KUKA KRL data list: pick_from_playingfield.dat

&ACCESS RV1
&REL 8
&PARAM DISKPATH = KRC:\R1\Program
DEFDAT  pick_from_playingfield PUBLIC

ENDDAT
